FUNCTION_BLOCK FB_SLITS_SCATTER EXTENDS FB_SLITS
VAR_INPUT
END_VAR
VAR_OUTPUT
END_VAR
VAR
END_VAR

ACT_init();
// Instantiate Function block for all the blades
ACT_Motion();
//SET and GET the requested and Actual values
ACT_CalculatePositions();

END_FUNCTION_BLOCK

(* stored: Version 1.1.0.1
   POU FB_SLITS_SCATTER: Id {e7865722-6c16-081f-3626-663de1d5af09}, SpecialFunc None *)
